FUNCTION_BLOCK FB_GripperRef
VAR_INPUT
END_VAR
VAR_OUTPUT
END_VAR
VAR
	nChannel 		: USINT;
	pToolCtrl		: POINTER TO BYTE;
	pToolState		: POINTER TO BYTE;
	bVialDetector	AT %I* : BOOL;
END_VAR

METHOD FB_init : BOOL
VAR_INPUT
	bInitRetains 	: BOOL; // if TRUE, the retain variables are initialized (warm start / cold start)
	bInCopyCode 	: BOOL;  // if TRUE, the instance afterwards gets moved into the copy code (online change)
	pMultiZRef 		: POINTER TO FB_MultiZRef;
END_VAR

VAR
	nFirstAdress : PVOID;
	nSelfAdress : PVOID;		
END_VAR
nFirstAdress := ADR(pMultiZRef^.aFbGripperRef);
nSelfAdress := THIS;
{IF hasvalue (RegisterSize, '32')}
nChannel := UDINT_TO_USINT((nSelfAdress - nFirstAdress)/SIZEOF(THIS^) + 1);
{ELSE}
nChannel := ULINT_TO_USINT((nSelfAdress - nFirstAdress)/SIZEOF(THIS^) + 1);
{END_IF}
pToolCtrl := ADR(pMultiZRef^.aFbZAxisRef[nChannel].stOutput.nToolCtrl);
pToolState := ADR(pMultiZRef^.aFbZAxisRef[nChannel].stInput.nToolState);
END_METHOD

METHOD M_Actuate
VAR_INPUT
	eCtrl : E_OpClCtrl;
END_VAR
pToolCtrl^ := eCtrl;
END_METHOD

PROPERTY P_bVialDetector : BOOL
GET
P_bVialDetector := NOT bVialDetector;
END_GET
END_PROPERTY

PROPERTY P_eGripperState : E_GripperState
GET
IF pToolState^ = 24 THEN
	P_eGripperState := E_GripperState.Open;
ELSIF pToolState^ = 9 THEN
	P_eGripperState := E_GripperState.HalfClosed;
ELSIF pToolState^ = 11 THEN
	P_eGripperState := E_GripperState.FullyClosed;
ELSE
	P_eGripperState := E_GripperState.Undefined;
END_IF
END_GET
END_PROPERTY

END_FUNCTION_BLOCK

(* stored: Version 1.1.0.1, ProductVersion 3.1.4024.6
   POU FB_GripperRef: Id {5ba6d2de-f4a7-4fba-8040-e12d05453dc1}, SpecialFunc None
   Method FB_init: Id {067f5934-8892-4b05-91db-878fa811ce39}
   Method M_Actuate: Id {debbd48d-4498-4f83-b798-dc89a925ac02}
   Property P_bVialDetector: Id {535017f4-4a94-44d8-bd5f-3698fbefa80b}
   Get Get: Id {8c0ba058-5935-40c3-a64a-7e6e8c91c7da}
   Property P_eGripperState: Id {b3b2a80e-cd6d-4623-bd52-e5ab2d84ab37}
   Get Get: Id {6699658c-ef1e-436b-a96e-b1e6f5716051} *)
